FUNCTION_BLOCK FB_AutoStartCoordinator
VAR_INPUT
    bRequest             : BOOL;  // WPF 的 bControlAuto 请求
    bCancel              : BOOL;  // Stop、Abort 或停止故障
    bHmiOnline           : BOOL;
    bControlAllowed      : BOOL;
    bGripperReady        : BOOL;
    bGripperActionFault  : BOOL;
    bProcessDone         : BOOL;  // 整套五盘流程已完成
    bTrayPlanCheckDone   : BOOL;  // Tray唯一来源：五层稳定检查完成
    bTrayPlanValid       : BOOL;
    bTrayPlanLocked      : BOOL;
    bTrayNoTrayAvailable : BOOL;
    tEnableTimeout       : TIME := GVL_SafetyConfig.stStartup.tEnableTimeout;
	bMachinePreparationDone  : BOOL;
	bMachinePreparationError : BOOL;
END_VAR

VAR_IN_OUT
    // 只读取轴状态；本 FB 不直接写轴命令。
    aAxes : ARRAY[1..GVL_Constants.cMaxAxisCount] OF ST_AxisInterface;
END_VAR

VAR_OUTPUT
    bTrayPlanRequest : BOOL;  // 准备后建立正式Plan；成功后保持至批次结束
    bTrayPlanChecking : BOOL; // 准备后的Plan检查；保持已准备轴使能
    bEnableAxes      : BOOL;  // MAIN 据此请求自动流程涉及的轴使能
    bProcessStart    : BOOL;  // 全部就绪后保持 TRUE，直到完成或中止
    bEnabling        : BOOL;  // 正在等待轴使能、就绪
    bStartRejected   : BOOL;  // 启动拒绝；准备后全无盘也沿用此语义
    bError           : BOOL;  // 启动阶段故障，保持供诊断
    bErrorPulse      : BOOL;  // 单周期脉冲，交给现有 Stop 链路
    bTimeout         : BOOL;
    uiErrorAxisIndex : UINT;  // 轴故障／超时对应的业务轴下标
    uiErrorCode      : UINT;  // 见实现区末尾的代码说明
	bMachinePreparationRequest : BOOL;// 保持型请求，直到整机准备完成。
END_VAR

VAR
    trigStart       : R_TRIG;
    fbEnableTimeout : TON;

    uiItem       : DINT;
    uiAxis       : UINT;
    bAllAxesReady : BOOL;

    eStep : E_AutoStartStep := E_AutoStartStep.Idle;
END_VAR

// 请求只受理上升沿，防止 WPF 长时间保持 TRUE 时重复启动。
trigStart(CLK := bRequest);

// TON 每个扫描周期调用一次。进入步骤 10 的下一周期开始计时。
fbEnableTimeout(
    IN := (eStep = E_AutoStartStep.WaitAxesReady) AND NOT bCancel,
    PT := tEnableTimeout
);

bErrorPulse := FALSE;

// Stop 优先级最高。本 FB 不撤轴使能：受控停止和掉使能
// 仍由 FB_AutoStopManager 按既有时序完成。
IF bCancel OR ((eStep = E_AutoStartStep.WaitTrayPlan) AND NOT bRequest) THEN
    eStep := E_AutoStartStep.Idle;
ELSE
    CASE eStep OF

        E_AutoStartStep.Idle: // 待机：只做一次启动准入检查
            IF trigStart.Q THEN
                bStartRejected := FALSE;
                bError := FALSE;
                bTimeout := FALSE;
                uiErrorAxisIndex := 0;
                uiErrorCode := TO_UINT(E_AutoStartErrorCode.None);

                IF NOT bHmiOnline THEN
                    bStartRejected := TRUE;
                    uiErrorCode := TO_UINT(E_AutoStartErrorCode.HmiOffline);

                ELSIF NOT bControlAllowed THEN
                    bStartRejected := TRUE;
                    uiErrorCode := TO_UINT(E_AutoStartErrorCode.ControlNotAllowed);

                ELSIF bGripperActionFault OR NOT bGripperReady THEN
                    bStartRejected := TRUE;
                    uiErrorCode := TO_UINT(E_AutoStartErrorCode.GripperNotReady);

                ELSE
                    // 在发使能之前确认八根参与轴均已配置。
                    FOR uiItem := LOWER_BOUND(GVL_AxisIndex.AutoProcessAxes, 1) TO UPPER_BOUND(GVL_AxisIndex.AutoProcessAxes, 1) DO
                        uiAxis := GVL_AxisIndex.AutoProcessAxes[uiItem];

                        IF NOT GVL_AxisConfig.AxisLimits[
                            uiAxis
                        ].bConfigured THEN
                            bStartRejected := TRUE;
                            uiErrorCode := TO_UINT(E_AutoStartErrorCode.AxisNotConfigured);
                            uiErrorAxisIndex := uiAxis;
                            EXIT;
                        END_IF;
                    END_FOR;

                    IF NOT bStartRejected THEN
                        // 基础准入后先使能、整机准备；此时绝不建立正式Plan。
                        eStep := E_AutoStartStep.WaitAxesReady;
                    END_IF;
                END_IF;
            END_IF;

        E_AutoStartStep.WaitTrayPlan:
            IF NOT bHmiOnline OR NOT bControlAllowed
                OR bGripperActionFault OR NOT bGripperReady THEN
                // 准备后只检查Plan，条件失效沿用启动拒绝。
                bStartRejected := TRUE;
                uiErrorCode := TO_UINT(E_AutoStartErrorCode.StartConditionLost);
                eStep := E_AutoStartStep.Idle;
            ELSIF bTrayPlanCheckDone THEN
                IF bTrayNoTrayAvailable THEN
                    // 全无盘仅StartRejected，不是Fault；MAIN撤销bControlAuto。
                    bStartRejected := TRUE;
                    uiErrorCode := TO_UINT(E_AutoStartErrorCode.NoTrayAvailable);
                    eStep := E_AutoStartStep.Idle;
                ELSIF bTrayPlanValid AND bTrayPlanLocked THEN
                    eStep := E_AutoStartStep.Running;
                END_IF;
            END_IF; // StableValid未全部成立时继续等待，不新增超时。

        E_AutoStartStep.WaitAxesReady: // 请求使能，读取 FB_AxisManager 上一扫描周期的轴状态
            IF NOT bHmiOnline
                OR NOT bControlAllowed
                OR bGripperActionFault
                OR NOT bGripperReady THEN

                bError := TRUE;
                bErrorPulse := TRUE;
                uiErrorCode := TO_UINT(E_AutoStartErrorCode.StartConditionLost);
                eStep := E_AutoStartStep.Idle;

            ELSE
                bAllAxesReady := TRUE;
                uiErrorAxisIndex := 0;

                FOR uiItem := LOWER_BOUND(GVL_AxisIndex.AutoProcessAxes, 1) TO UPPER_BOUND(GVL_AxisIndex.AutoProcessAxes, 1) DO
                    uiAxis := GVL_AxisIndex.AutoProcessAxes[uiItem];

                    IF aAxes[uiAxis].Alarm.bError THEN
                        bError := TRUE;
                        bErrorPulse := TRUE;
                        uiErrorCode := TO_UINT(E_AutoStartErrorCode.AxisAlarm);
                        uiErrorAxisIndex := uiAxis;
                        eStep := E_AutoStartStep.Idle;
                        EXIT;
                    END_IF;

                    IF NOT aAxes[uiAxis].State.bReady THEN
                        bAllAxesReady := FALSE;

                        // 保留第一根未就绪轴，供超时诊断。
                        IF uiErrorAxisIndex = 0 THEN
                            uiErrorAxisIndex := uiAxis;
                        END_IF;
                    END_IF;
                END_FOR;

                IF NOT bErrorPulse THEN
					IF bAllAxesReady THEN
						uiErrorAxisIndex := 0;
						eStep := E_AutoStartStep.WaitMachinePreparation;
                    ELSIF fbEnableTimeout.Q THEN
                        bError := TRUE;
                        bTimeout := TRUE;
                        bErrorPulse := TRUE;
                        uiErrorCode := TO_UINT(E_AutoStartErrorCode.AxisReadyTimeout);
                        eStep := E_AutoStartStep.Idle;
                    END_IF;
                END_IF;
            END_IF;

		E_AutoStartStep.WaitMachinePreparation:
			IF bMachinePreparationError THEN
				// 整机准备故障由MachineSupervisor统一锁存。
				eStep := E_AutoStartStep.Idle;
		
			ELSIF bMachinePreparationDone THEN
				eStep := E_AutoStartStep.WaitTrayPlan;
			END_IF;

        E_AutoStartStep.Running: // 保持启动许可；现有流程 FB 自己锁存 bStart 上升沿
            IF bProcessDone THEN
                eStep := E_AutoStartStep.Idle;
            END_IF;

        ELSE
            bError := TRUE;
            bErrorPulse := TRUE;
            uiErrorCode := TO_UINT(E_AutoStartErrorCode.InvalidProcessStep);
            eStep := E_AutoStartStep.Idle;
    END_CASE;
END_IF;

// 统一从状态机导出输出，避免 Stop 同一扫描仍下发启动。
// 根据本周期最终状态发布输出；Stop 时三个输出立即撤销。
// 计划请求贯穿本轮生命周期，Tray据此冻结/释放唯一计划。
bTrayPlanChecking := (eStep = E_AutoStartStep.WaitTrayPlan);
// Preparation之前保持FALSE；唯一计划仅在准备完成后建立。
bTrayPlanRequest := bTrayPlanChecking
    OR (eStep = E_AutoStartStep.Running);

bEnabling :=
    bTrayPlanChecking
    OR (eStep = E_AutoStartStep.WaitAxesReady)
    OR
    (eStep = E_AutoStartStep.WaitMachinePreparation);

// WaitMachinePreparation期间使能权属于PreparationCmd，
// 不再继续写入无权的AutoCmd。
bEnableAxes :=
    (eStep = E_AutoStartStep.WaitAxesReady)
    OR
    (eStep = E_AutoStartStep.Running);
	
bMachinePreparationRequest :=
    (eStep = E_AutoStartStep.WaitMachinePreparation);

bProcessStart :=
    (eStep = E_AutoStartStep.Running);

END_FUNCTION_BLOCK

(* stored: Version 1.1.0.1, ProductVersion 3.1.4026.20
   POU FB_AutoStartCoordinator: Id {d00eb36f-61db-4727-88b2-be6ec64efbc0}, SpecialFunc None *)
